Yaskawa INFORM job: 01-SAFETY.JBI

/JOB
//NAME 01-SAFETY
///FOLDERNAME SAFETY
//POS
///NPOS 1,1,0,0,0,0
///TOOL 0
///POSTYPE ROBOT
///RECTAN
///RCONF 0,0,0,0,0,0,0,0,0,0,0,0,0,0,0,0,0,0,0,0,0,0,0,0
C00000=1043.305,21.307,-685.481,-3.2772,-33.1507,3.6069
BC00000=539.760,5648.937,840.904
//INST
///DATE 2023/07/13 09:20
///ATTR SC,RW,RJ
////FRAME ROBOT
///GROUP1 RB1,BS1
NOP
*START
MOVJ C00000 BC00000 VJ=20.00
JUMP *START
END
